SUBAPPLICATION VT_active (* Subapplication Type *)
  (* Standard: 61499-2 *)
  (* Version 1.0, 2023-02-19, franz *)
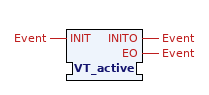
  EVENT_INPUT
    INIT;
  END_EVENT
  EVENT_OUTPUT
    INITO;
    EO;
  END_EVENT
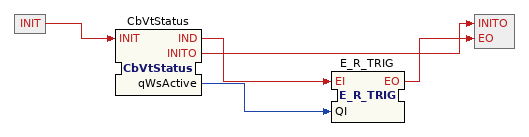
  FBS
    E_R_TRIG : E_R_TRIG;
    CbVtStatus : CbVtStatus;
  END_FBS
  EVENT_CONNECTIONS
    E_R_TRIG.EO TO EO;
    CbVtStatus.IND TO E_R_TRIG.EI;
    CbVtStatus.INITO TO INITO;
    INIT TO CbVtStatus.INIT;
  END_CONNECTIONS
  DATA_CONNECTIONS
    CbVtStatus.qWsActive TO E_R_TRIG.QI;
  END_CONNECTIONS
END_SUBAPPLICATION
